// TwinCAT 3 PLC project FSM
// ProgramVersion: 3.1.4026.18
// libraries:
//   Tc2_EtherCAT, * (Beckhoff Automation GmbH)
//   Tc2_Standard, * (Beckhoff Automation GmbH)
//   Tc2_System, * (Beckhoff Automation GmbH)
//   TcUnit, * (www.tcunit.org)
// project tree:
//   DUTs/ E_Command.TcDUT (not stored), E_PodState.TcDUT (not stored)
//   GVLs/ GVL_FSM.TcGVL, GVL_Levi.TcGVL (not stored), GVL_Prop.TcGVL (not stored), GVL_PT.TcGVL
//   / PlcTask.TcTTO (not stored)
//   POUs/Fsm/ BasicChecks.TcPOU (not stored), CheckCritical.TcPOU, FB_Charge.TcPOU (not stored), FB_Discharge.TcPOU, FB_Handle_Emergency.TcPOU, Handle_Movement.TcPOU, Main_FSM.TcPOU
//   POUs/ MAIN.TcPOU
//   POUs/Tests/ FB_Test_FSM.TcPOU
// real-time tasks:
//   TASK PlcTask: cycle T#10ms, priority 20, ADS port 350
//   TASK HeartBeat: cycle T#10ms, priority 1, ADS port 351

// ---- GVLs/GVL_FSM.TcGVL
{attribute 'qualified_only'}
VAR_GLOBAL
	enable_heartbeat:		BOOL;
	heartbeat_OK: 			BOOL;
	precharge:				BOOL;
	engage_brakes:			BOOL;
	brakes_engaged:			BOOL;
	enable_levi_checks: 	BOOL;
	enable_prop_checks: 	BOOL;
	enable_temp_checks: 	BOOL;
	safety_inputs_valid: 	BOOL;
	can_bus_ok: 			BOOL;
	ethercat_ready: 		BOOL;
	sdc_closed: 			BOOL;
	critical_temp: 			INT;
	open_SDC: 				BOOL	:= TRUE;
	enable_telemetry: BOOL;
	enable_PT_checks: BOOL;
	trigger_EL: BOOL;
END_VAR

// ---- GVLs/GVL_PT.TcGVL
{attribute 'qualified_only'}
VAR_GLOBAL
	HVAL_STATUS:			USINT;
	ERROR_STATUS: 			USINT;
	MAX_TEMP: 				UINT;
	emergency_shutdown: 	BOOL;
	total_voltage: UINT;
END_VAR

// ---- POUs/Fsm/CheckCritical.TcPOU
FUNCTION CheckCritical : BOOL
VAR_INPUT
END_VAR
VAR
END_VAR

CheckCritical := 
    NOT GVL_FSM.sdc_closed OR
    GVL_PT.ERROR_STATUS <> 0 OR
    GVL_PT.MAX_TEMP > GVL_FSM.critical_temp OR
    GVL_Levi.levitation_fault OR
    GVL_Prop.propulsion_fault;

END_FUNCTION

// ---- POUs/Fsm/FB_Discharge.TcPOU
FUNCTION_BLOCK FB_Discharge
VAR_INPUT
END_VAR
VAR_OUTPUT
END_VAR
VAR
END_VAR

END_FUNCTION_BLOCK

// ---- POUs/Fsm/FB_Handle_Emergency.TcPOU
FUNCTION_BLOCK FB_Handle_Emergency
VAR_INPUT
    execute: 				BOOL;
END_VAR
VAR_OUTPUT
    busy: 					BOOL;
END_VAR
VAR
    state: 					INT := 0;
    tonDelay: 				TON;
	allActionsComplete:		BOOL;
END_VAR

IF NOT execute THEN
    state := 0;
    busy := FALSE;
    tonDelay(IN := FALSE);
    RETURN;
END_IF

busy := TRUE;
CASE state OF
    0:  GVL_FSM.trigger_EL := TRUE;
		GVL_FSM.open_SDC := TRUE;
        GVL_FSM.engage_brakes := TRUE;
        GVL_Prop.propulsion_enable := FALSE;
        GVL_Levi.levitation_active := FALSE;
        GVL_PT.emergency_shutdown := TRUE;
        state := 1;
        
    1:  allActionsComplete := 
            NOT GVL_FSM.sdc_closed AND
            GVL_FSM.brakes_engaged AND
            NOT GVL_Prop.propulsion_active AND
            NOT GVL_Levi.levitation_active;
        
        IF allActionsComplete THEN
            state := 2;
        END_IF
        
    2:	tonDelay(IN := TRUE, PT := T#200MS);
        IF tonDelay.Q THEN
			GVL_FSM.trigger_EL := FALSE;
            busy := FALSE;
			execute := FALSE;
        END_IF
END_CASE

END_FUNCTION_BLOCK

// ---- POUs/Fsm/Handle_Movement.TcPOU
FUNCTION Handle_Movement : BOOL
VAR_INPUT
END_VAR
VAR
END_VAR

END_FUNCTION

// ---- POUs/Fsm/Main_FSM.TcPOU
FUNCTION_BLOCK Main_FSM

VAR_INPUT
	currentCmd:					E_Command 	:= E_Command.CMD_NONE;
END_VAR


VAR_OUTPUT
	currentState: 				E_PodState  := E_PodState.STATE_BOOT;
END_VAR

VAR
	criticalFault:				BOOL;
	charging_in_progress:		BOOL;
	discharging_in_progress:	BOOL;
	
	fb_handle_emergency:		FB_Handle_Emergency;
	fb_discharge:				FB_Discharge;
	fb_charge:					FB_Charge;
END_VAR

IF currentCmd = E_Command.CMD_EMERGENCY OR (CheckCritical() AND currentState >= 4) THEN
	currentState := E_PodState.STATE_EMERGENCY;
	criticalFault := TRUE;
	FB_Handle_Emergency();
ELSIF currentState = E_PodState.STATE_MOVEMENT AND 
    GVL_Prop.speed = 0 AND GVL_Prop.target_speed = 0 THEN
		currentState := E_PodState.STATE_LEVITATION;
ELSIF currentState = E_PodState.STATE_DEMO AND GVL_FSM.brakes_engaged THEN
    currentState := E_PodState.STATE_EMERGENCY;
ELSIF currentState = E_PodState.STATE_BOOT AND BasicChecks() THEN
	currentState := E_PodState.STATE_SYNC;
END_IF

CASE currentState OF
	E_PodState.STATE_EMERGENCY:
		IF criticalFault THEN
			FB_Handle_Emergency();
		ELSIF currentCmd = E_Command.CMD_TO_MAINTENANCE THEN
			GVL_FSM.engage_brakes := FALSE;
			currentState := E_PodState.STATE_MAINTENANCE;
		END_IF
		
	E_PodState.STATE_BOOT:  
		IF BasicChecks() THEN
			currentState := E_PodState.STATE_SYNC;
		END_IF
		
	E_PodState.STATE_SYNC:
		GVL_FSM.enable_heartbeat := TRUE;
		IF GVL_FSM.heartbeat_OK AND currentCmd = E_Command.CMD_TO_IDLE THEN
			currentState := E_PodState.STATE_IDLE;
		END_IF
		
	E_PodState.STATE_IDLE:
		// maybe basic checks again WC state - 8
		GVL_FSM.enable_PT_checks := TRUE;
		GVL_FSM.enable_temp_checks := TRUE;
		GVL_FSM.enable_telemetry := TRUE;
		
		IF currentCmd = E_Command.CMD_TO_HV_ACTIVE THEN
			FB_Charge();
			IF GVL_PT.HVAL_STATUS = 1 AND GVL_PT.total_voltage >= 550 THEN
				currentState := E_PodState.STATE_HV_ACTIVE;
			END_IF
		ELSIF currentCmd = E_Command.CMD_TO_MAINTENANCE THEN
			GVL_FSM.engage_brakes := FALSE;
			currentState := E_PodState.STATE_MAINTENANCE;
		END_IF
		
	E_PodState.STATE_HV_ACTIVE:
		GVL_FSM.enable_levi_checks := TRUE;
		GVL_FSM.enable_prop_checks := TRUE;
				
		IF currentCmd = E_Command.CMD_TO_DEMO AND NOT CheckCritical() THEN
			GVL_FSM.engage_brakes := FALSE;
			currentState := E_PodState.STATE_DEMO;
		ELSIF currentCmd = E_Command.CMD_TO_IDLE THEN
			GVL_FSM.open_SDC := TRUE;
			FB_Discharge();
			IF GVL_PT.HVAL_STATUS = 0 AND GVL_Levi.drive_voltages = 0 AND GVL_Prop.drive_voltages = 0 THEN
				currentState := E_PodState.STATE_IDLE;
			END_IF
		END_IF
		
	E_PodState.STATE_DEMO:
		IF currentCmd = E_Command.CMD_TO_IDLE THEN
			GVL_FSM.engage_brakes := TRUE;
			GVL_FSM.open_SDC := TRUE;
			FB_Discharge();
			IF GVL_FSM.brakes_engaged AND GVL_PT.HVAL_STATUS = 0 THEN
				currentState := E_PodState.STATE_IDLE;
			END_IF
		ELSIF currentCmd = E_Command.CMD_TO_LEVITATION THEN
			GVL_Levi.levitation_active := TRUE;
			currentState := E_PodState.STATE_LEVITATION;
		END_IF
		
	E_PodState.STATE_LEVITATION:
		IF currentCmd = E_Command.CMD_TO_DEMO THEN
			GVL_Levi.levitation_active := FALSE;
			currentState := E_PodState.STATE_DEMO;
		ELSIF currentCmd = E_Command.CMD_TO_MOVEMENT THEN
			currentState := E_PodState.STATE_MOVEMENT;
			Handle_movement();
		END_IF
		
	E_PodState.STATE_MOVEMENT:
		Handle_movement();
		
	E_PodState.STATE_MAINTENANCE:
		IF currentCmd = E_Command.CMD_TO_IDLE THEN
			GVL_FSM.engage_brakes := TRUE;
			IF GVL_FSM.brakes_engaged THEN
				currentState := E_PodState.STATE_IDLE;
			END_IF
		END_IF
		
END_CASE

END_FUNCTION_BLOCK

// ---- POUs/MAIN.TcPOU
PROGRAM MAIN
VAR
	main_fsm	: Main_FSM;
	main_tests	: FB_Test_FSM;
	
	tests_on	: BOOL	:= TRUE;
END_VAR

IF tests_on THEN
	TcUnit.RUN();
ELSE
	main_fsm();
END_IF

END_PROGRAM

// ---- POUs/Tests/FB_Test_FSM.TcPOU
FUNCTION_BLOCK FB_Test_FSM EXTENDS TcUnit.FB_TestSuite
VAR_INPUT
END_VAR
VAR_OUTPUT
END_VAR
VAR
END_VAR

END_FUNCTION_BLOCK
